# EPICS autosave request: m-epics-ADKafka/ADKafkaApp/Db/ADKafka.req
# Nothing extra needed beyond NDPluginBase_settings.req for now
file "ADBase_settings.req", P=$(P), R=$(R)
